// TIA Portal V17 export
// export: Created 2024-09-02T12:50:20.4107837Z, ExportSetting WithDefaults, DisplayName Totally Integrated Automation Portal, DisplayVersion V17, DisplayName TIA Portal Openness, DisplayVersion V17, DisplayName TIA Portal Version Control Interface, DisplayVersion V17, DisplayName STEP 7 Professional, DisplayVersion V17, DisplayName STEP 7 Safety, DisplayVersion V17, DisplayName WinCC Professional, DisplayVersion V17
DATA_BLOCK "MdsDB1_FG02_Data_SLG3_OP70"   // DB1111
{ S7_Optimized_Access := 'FALSE'; DB_Accessible_From_OPC_UA := 'FALSE' }
VERSION : 0.1
// stored: AutoNumber false, DBAccessibleFromOPCUA false, IsOnlyStoredInLoadMemory false, IsWriteProtectedInAS false
   VAR
      read : Struct
         General { S7_SetPoint := 'True'} : "typ_General";
         Station : Struct
            OP10 : "OP10";
            OP20 : "OP20";
            OP30 { S7_SetPoint := 'True'} : "OP30";
            OP40 : "OP40";
            OP50 : "OP50";
            OP60 : "OP60";
            OP70_1 : "OP701";
            OP70_2 : "OP702";
            OP70_3 : "OP703";
         END_STRUCT;
      END_STRUCT;
      write : Struct
         General { S7_SetPoint := 'True'} : "typ_General";
         Station : Struct
            OP10 : "OP10";
            OP20 : "OP20";
            OP30 { S7_SetPoint := 'True'} : "OP30";
            OP40 : "OP40";
            OP50 : "OP50";
            OP60 : "OP60";
            OP70_1 : "OP701";
            OP70_2 : "OP702";
            OP70_3 : "OP703";
         END_STRUCT;
      END_STRUCT;
      init : Struct
         General { S7_SetPoint := 'True'} : "typ_General";
         Station : Struct
            OP10 : "OP10";
            OP20 : "OP20";
            OP30 { S7_SetPoint := 'True'} : "OP30";
            OP40 : "OP40";
            OP50 : "OP50";
            OP60 : "OP60";
            OP70_1 : "OP701";
            OP70_2 : "OP702";
            OP70_3 : "OP703";
         END_STRUCT;
      END_STRUCT;
   END_VAR
BEGIN
END_DATA_BLOCK
